FUNCTION Scaling : REAL
VAR_INPUT
	Input : INT;
	Imin : REAL;
	Imax : REAL;
	Qmin : REAL;
	Qmax : REAL;
END_VAR
VAR_OUTPUT
END_VAR
VAR
	schaalfactor : REAL;
	offset : REAL;
END_VAR

schaalfactor := (Qmax - Qmin)/(Imax - Imin);
offset := Qmin - (Imin*schaalfactor);
Scaling := (schaalfactor * Input + offset);

END_FUNCTION

(* stored: Version 1.1.0.1, ProductVersion 3.1.4024.3
   POU Scaling: Id {66bf3739-5431-4fc7-96ca-4ae20f49e9c6}, SpecialFunc None *)
